// TwinCAT 3 PLC project Untitled1
// ProgramVersion: 3.1.4026.16
// libraries:
//   Recipe Management, * (System)
//   Tc2_Standard, * (Beckhoff Automation GmbH)
//   Tc2_System, * (Beckhoff Automation GmbH)
//   Tc3_Module, * (Beckhoff Automation GmbH)
// project tree:
//   DUTs/ dt_params.TcDUT
//   / PlcTask.TcTTO, RecipeManager.TcRMO (not stored), RecipeTask.TcTTO
//   POUs/ MAIN.TcPOU, Recipes.TcPOU
// real-time tasks:
//   TASK PlcTask: cycle T#10ms, priority 6, ADS port 350
//   TASK RecipeTask: cycle T#100000us, priority 8, ADS port 351

CONFIGURATION Untitled1
    RESOURCE PLC ON TwinCAT3
        TASK PlcTask(INTERVAL := T#10ms, PRIORITY := 6);
        TASK RecipeTask(INTERVAL := T#100000us, PRIORITY := 8);
        PROGRAM MAIN WITH PlcTask : MAIN;
        PROGRAM Recipes WITH RecipeTask : Recipes;
    END_RESOURCE
END_CONFIGURATION

// ---- DUTs/dt_params.TcDUT
TYPE dt_params :
STRUCT
	scale	: LREAL;
	offset	: LREAL;
	f		: WORD;
END_STRUCT
END_TYPE

// ---- POUs/MAIN.TcPOU
PROGRAM MAIN
VAR
	var1	: UINT;
	var2	: LREAL;
	var3	: STRING;
	var4	: BOOL;
	var5	: ARRAY[0..999] OF T_MaxString;
	var6	: ARRAY[0..2] OF dt_params;

END_VAR


//just commands to the slow task
recipes.load;
recipes.save;
recipes.count;
recipes.delete;
recipes.name;
recipes.result;

END_PROGRAM

// ---- POUs/Recipes.TcPOU
PROGRAM Recipes
VAR_INPUT
	save	: BOOL;
	load	: BOOL;
	delete	: BOOL;
	count	: BOOL;
	name	: T_MaxString;
END_VAR
VAR_OUTPUT
	result	: DWORD;
END_VAR
VAR
	reci	: RecipeManCommands;
END_VAR
VAR CONSTANT
	defname	: T_MaxString := 'testing123';
END_VAR



IF save THEN
	save := FALSE;
	result := reci.CreateRecipe(defname, name);
END_IF

IF load THEN
	load := FALSE;
	result := reci.LoadAndWriteRecipe(defname, name);
END_IF

IF delete THEN
	delete := FALSE;
	result := reci.DeleteRecipe(defname, name);
END_IF

IF count THEN
	count := FALSE;
	result := INT_TO_DWORD(reci.GetRecipeCount(defname));
END_IF

END_PROGRAM
